// TIA Portal V18 export
FUNCTION_BLOCK "FPDRxMonitorTwoEncodersFB"   // FB63, FBD
{ S7_Optimized_Access := 'TRUE' }
VERSION : 0.1
// stored: AutoNumber true, IsIECCheckEnabled false, IsRetainMemResEnabled false, MemoryReserve 100, SetENOAutomatically false, UDAEnableTagReadback false
   VAR_INPUT
      pos1 { ExternalAccessible := 'False'; ExternalVisible := 'False'; ExternalWritable := 'False'} : Real;
      pos2 { ExternalAccessible := 'False'; ExternalVisible := 'False'; ExternalWritable := 'False'} : Real;
      allowedDelta { ExternalAccessible := 'False'; ExternalVisible := 'False'; ExternalWritable := 'False'} : Real;
      pt : Time;
   END_VAR
   VAR_OUTPUT
      error { ExternalAccessible := 'False'; ExternalVisible := 'False'; ExternalWritable := 'False'} : Bool;
   END_VAR
   VAR
      tonER { S7_SetPoint := 'True'} : TON_TIME;
   END_VAR
   VAR_TEMP
      deltaDangerous : Bool;
   END_VAR
BEGIN

REGION Network 2 (SCL)
   #deltaDangerous := ABS(#pos2 - #pos1)> #allowedDelta;
END_REGION

REGION Network 3
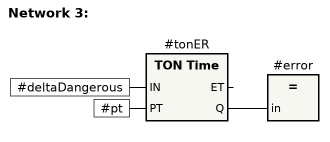
   #tonER(IN := #deltaDangerous, PT := #pt);   // TON
   #error := #tonER.Q;
END_REGION
END_FUNCTION_BLOCK
